// TIA Portal V20 export
TYPE "LER_TypeFATMode_HoursTest_SetValue"
// stored: Access Published
   STRUCT
      SelectHours_SetValue : Time_Of_Day;
   END_STRUCT;
END_TYPE
